TYPE ELL9AttenuationFilterConfig EXTENDS DeviceConfiguration :
STRUCT
	SerialCommunication : SerialCommunication;
END_STRUCT
END_TYPE

(* stored: Version 1.1.0.1, ProductVersion 3.1.4024.4
   DUT ELL9AttenuationFilterConfig: Id {67c65185-f6b7-4b72-a2a4-9a84e25601c4} *)
